FUNCTION S_Scale : DINT
VAR_INPUT
	nAnalogInput : DINT;
END_VAR
VAR
END_VAR

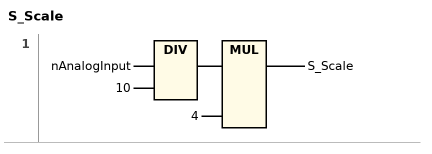
// NETWORK 1
S_Scale := (nAnalogInput / 10) * 4;

END_FUNCTION

(* stored: Version 1.1.0.1, ProductVersion 3.1.4024.0
   POU S_Scale: Id {641cc4ea-6338-475f-b3ca-8aca85ced253}, SpecialFunc None *)
